	UF : 1, UT : 1,		CONFIG : 'N U T, 0, 0, 0',
	X =   648.092  mm,	Y = -1312.832  mm,	Z =  1599.443  mm,
	W =   -41.810 deg,	P =   -20.894 deg,	R =   -21.724 deg
   GP2:
	UF : 0, UT : 1,
	J1=   180.000 deg,	J2=   -90.000 deg
};
P[708]{
   GP1:
	UF : 1, UT : 1,		CONFIG : 'N U T, 0, 0, 0',
	X =   973.093  mm,	Y =   -11.831  mm,	Z =  2176.445  mm,
	W =     -.010 deg,	P =   -45.000 deg,	R =     0.000 deg
   GP2:
	UF : 0, UT : 1,
	J1=   180.000 deg,	J2=    90.000 deg
};
P[709]{
   GP1:
	UF : 1, UT : 1,		CONFIG : 'N U T, 0, 0, 0',
	X =  1331.092  mm,	Y =   987.169  mm,	Z =  1342.444  mm,
	W =     -.010 deg,	P =    45.000 deg,	R =   -90.000 deg
   GP2:
	UF : 0, UT : 1,
	J1=   180.000 deg,	J2=    90.000 deg
};
P[710]{
   GP1:
	UF : 1, UT : 1,		CONFIG : 'N U T, 0, 0, 0',
	X =  1864.092  mm,	Y =  1212.638  mm,	Z =  1342.445  mm,
	W =    44.958 deg,	P =    -2.212 deg,	R =     2.229 deg
   GP2:
	UF : 0, UT : 1,
	J1=   180.000 deg,	J2=    90.000 deg
};
P[711]{
   GP1:
	UF : 1, UT : 1,		CONFIG : 'N U T, 0, 0, 0',
	X =  1940.973  mm,	Y =  1347.132  mm,	Z =  1061.188  mm,
	W =    41.277 deg,	P =    19.800 deg,	R =   -21.086 deg
   GP2:
	UF : 0, UT : 1,
	J1=   180.000 deg,	J2=    90.000 deg
};
P[712]{
   GP1:
	UF : 1, UT : 1,		CONFIG : 'N U T, 0, 0, 0',
	X =  1901.875  mm,	Y =  1465.160  mm,	Z =  1036.238  mm,
	W =    41.263 deg,	P =    19.805 deg,	R =   -17.225 deg
   GP2:
	UF : 1, UT : 1,
	J1=   180.000 deg,	J2=    90.000 deg
};
P[713]{
   GP1:
	UF : 1, UT : 1,		CONFIG : 'N U T, 0, 0, 0',
	X =  1934.116  mm,	Y =  1464.614  mm,	Z =  1037.732  mm,
	W =    41.277 deg,	P =    19.801 deg,	R =   -17.230 deg
   GP2:
	UF : 1, UT : 1,
	J1=   180.000 deg,	J2=    90.000 deg
};
P[714]{
   GP1:
	UF : 1, UT : 1,		CONFIG : 'N U T, 0, 0, 0',
	X =  1965.909  mm,	Y =  1468.963  mm,	Z =  1032.171  mm,
	W =    41.272 deg,	P =    19.803 deg,	R =   -17.223 deg
   GP2:
	UF : 1, UT : 1,
	J1=   180.000 deg,	J2=    90.000 deg
};
P[715]{
   GP1:
	UF : 1, UT : 1,		CONFIG : 'N U T, 0, 0, 0',
	X =  1996.605  mm,	Y =  1480.121  mm,	Z =  1030.618  mm,
	W =    41.277 deg,	P =    19.801 deg,	R =     6.735 deg
   GP2:
	UF : 1, UT : 1,
	J1=   180.000 deg,	J2=    90.000 deg
};
P[716]{
   GP1:
	UF : 1, UT : 1,		CONFIG : 'N U T, 0, 0, 0',
	X =  1999.792  mm,	Y =  1488.994  mm,	Z =  1027.439  mm,
	W =    43.863 deg,	P =    11.272 deg,	R =    16.919 deg
   GP2:
	UF : 1, UT : 1,
	J1=   180.000 deg,	J2=    90.000 deg
};
P[717]{
   GP1:
	UF : 1, UT : 1,		CONFIG : 'N U T, 0, 0, 0',
	X =  2007.580  mm,	Y =  1422.903  mm,	Z =  1059.661  mm,
	W =    44.305 deg,	P =     8.850 deg,	R =     3.803 deg
   GP2:
	UF : 1, UT : 1,
	J1=   180.000 deg,	J2=    90.000 deg
};
P[718]{
   GP1:
	UF : 1, UT : 1,		CONFIG : 'N U T, 0, 0, 0',
	X =  1864.092  mm,	Y =  1212.638  mm,	Z =  1342.444  mm,
	W =    44.958 deg,	P =    -2.212 deg,	R =     2.229 deg
   GP2:
	UF : 0, UT : 1,
	J1=   180.000 deg,	J2=    90.000 deg
};
P[729]{
   GP1:
	UF : 1, UT : 1,		CONFIG : 'F U T, 0, 0, 0',
	X =   818.947  mm,	Y =   972.802  mm,	Z =  1108.910  mm,
	W =    50.730 deg,	P =      .639 deg,	R =   -51.736 deg
   GP2:
	UF : 1, UT : 1,
	J1=   180.000 deg,	J2=   150.000 deg
};
P[730]{
   GP1:
	UF : 1, UT : 1,		CONFIG : 'F U T, 0, 0, 0',
	X =  1078.589  mm,	Y =   991.016  mm,	Z =  1063.910  mm,
	W =    50.730 deg,	P =      .639 deg,	R =   -51.736 deg
   GP2:
	UF : 1, UT : 1,
	J1=   180.000 deg,	J2=   150.000 deg
};
P[731]{
   GP1:
	UF : 1, UT : 1,		CONFIG : 'F U T, 0, 0, 0',
	X =  1104.853  mm,	Y =  1006.203  mm,	Z =  1025.639  mm,
	W =    44.130 deg,	P =    -6.203 deg,	R =   -51.549 deg
   GP2:
	UF : 1, UT : 1,
	J1=   180.000 deg,	J2=   150.000 deg
};
P[732]{
   GP1:
	UF : 1, UT : 1,		CONFIG : 'F U T, 0, 0, 0',
	X =  1114.844  mm,	Y =  1000.704  mm,	Z =  1027.080  mm,
	W =    43.014 deg,	P =    -7.268 deg,	R =   -34.946 deg
   GP2:
	UF : 1, UT : 1,
	J1=   180.000 deg,	J2=   150.000 deg
};
P[733]{
   GP1:
	UF : 1, UT : 1,		CONFIG : 'F U T, 0, 0, 0',
	X =  1125.597  mm,	Y =   997.219  mm,	Z =  1027.206  mm,
	W =    42.651 deg,	P =   -14.126 deg,	R =   -20.722 deg
   GP2:
	UF : 1, UT : 1,
	J1=   180.000 deg,	J2=   150.000 deg
};
P[734]{
   GP1:
	UF : 1, UT : 1,		CONFIG : 'F U T, 0, 0, 0',
	X =  1138.321  mm,	Y =   996.177  mm,	Z =  1027.210  mm,
	W =    42.651 deg,	P =   -14.126 deg,	R =   -27.080 deg
   GP2:
	UF : 1, UT : 1,
	J1=   180.000 deg,	J2=   150.000 deg
};
P[735]{
   GP1:
	UF : 1, UT : 1,		CONFIG : 'F U T, 0, 0, 0',
	X =  1090.032  mm,	Y =   963.970  mm,	Z =  1058.684  mm,
	W =    50.535 deg,	P =   -23.426 deg,	R =   -25.981 deg
   GP2:
	UF : 1, UT : 1,
	J1=   180.000 deg,	J2=   150.000 deg
};
P[736]{
   GP1:
	UF : 1, UT : 1,		CONFIG : 'F U T, 0, 0, 0',
	X =   866.460  mm,	Y =   968.970  mm,	Z =  1058.684  mm,
	W =    50.535 deg,	P =   -23.426 deg,	R =   -25.981 deg
   GP2:
	UF : 1, UT : 1,
	J1=   180.000 deg,	J2=   150.000 deg
};
P[737]{
   GP1:
	UF : 1, UT : 1,		CONFIG : 'F U T, 0, 0, 0',
	X =   866.460  mm,	Y =   968.969  mm,	Z =  1794.399  mm,
	W =    50.535 deg,	P =   -23.425 deg,	R =   -25.981 deg
   GP2:
	UF : 1, UT : 1,
	J1=   180.000 deg,	J2=   150.000 deg
};
P[749]{
   GP1:
	UF : 1, UT : 1,		CONFIG : 'N U B, 0, 0, 0',
	X =   361.637  mm,	Y =   -13.715  mm,	Z =  2427.062  mm,
	W =     -.019 deg,	P =   -39.997 deg,	R =      .013 deg
   GP2:
	UF : 1, UT : 1,
	J1=   100.000 deg,	J2=   -90.000 deg
};
P[750]{
   GP1:
	UF : 1, UT : 1,		CONFIG : 'N U T, 0, 0, 0',
	X =   345.640  mm,	Y = -1572.170  mm,	Z =  1050.335  mm,
	W =    56.087 deg,	P =     8.668 deg,	R =   -95.934 deg
   GP2:
	UF : 1, UT : 1,
	J1=   100.000 deg,	J2=   -90.000 deg
};
P[751]{
   GP1:
	UF : 1, UT : 1,		CONFIG : 'N U T, 0, 0, -1',
	X =  2515.039  mm,	Y = -1508.170  mm,	Z =  1050.334  mm,
	W =   -50.284 deg,	P =   -30.325 deg,	R =    67.097 deg
   GP2:
	UF : 0, UT : 1,
	J1=   100.000 deg,	J2=   -90.000 deg
};
P[752]{
   GP1:
	UF : 1, UT : 1,		CONFIG : 'N U T, 0, 0, 0',
	X =  2788.736  mm,	Y = -1483.274  mm,	Z =   933.541  mm,
	W =   -37.771 deg,	P =   -31.405 deg,	R =    42.828 deg
   GP2:
	UF : 1, UT : 1,
	J1=   100.000 deg,	J2=   -90.000 deg
};
P[753]{
   GP1:
	UF : 1, UT : 1,		CONFIG : 'N U T, 0, 0, 0',
	X =  2790.127  mm,	Y = -1512.097  mm,	Z =   933.343  mm,
	W =   -37.782 deg,	P =   -31.394 deg,	R =    42.842 deg
   GP2:
	UF : 1, UT : 1,
	J1=   100.000 deg,	J2=   -90.000 deg
};
P[754]{
   GP1:
	UF : 1, UT : 1,		CONFIG : 'N U T, 0, 0, 0',
	X =  2777.828  mm,	Y = -1541.019  mm,	Z =   932.405  mm,
	W =   -42.870 deg,	P =   -22.985 deg,	R =    39.985 deg
   GP2:
	UF : 1, UT : 1,
	J1=   100.000 deg,	J2=   -90.000 deg
};
P[755]{
   GP1:
	UF : 1, UT : 1,		CONFIG : 'N U T, 0, 0, 0',
	X =  2762.396  mm,	Y = -1555.396  mm,	Z =   929.477  mm,
	W =   -45.718 deg,	P =   -14.892 deg,	R =    35.274 deg
   GP2:
	UF : 1, UT : 1,
	J1=   100.000 deg,	J2=   -90.000 deg
};
P[756]{
   GP1:
	UF : 1, UT : 1,		CONFIG : 'N U T, 0, 0, 0',
	X =  2731.844  mm,	Y = -1574.335  mm,	Z =   920.084  mm,
	W =   -45.718 deg,	P =   -14.891 deg,	R =    30.406 deg
   GP2:
	UF : 1, UT : 1,
	J1=   100.000 deg,	J2=   -90.000 deg
};
P[757]{
   GP1:
	UF : 1, UT : 1,		CONFIG : 'N U T, 0, 0, 0',
	X =  2725.103  mm,	Y = -1575.819  mm,	Z =   919.847  mm,
	W =   -45.718 deg,	P =   -14.891 deg,	R =    18.309 deg
   GP2:
	UF : 1, UT : 1,
	J1=   100.000 deg,	J2=   -90.000 deg
};
P[758]{
   GP1:
	UF : 1, UT : 1,		CONFIG : 'N U T, 0, 0, 0',
	X =  2712.522  mm,	Y = -1579.347  mm,	Z =   916.110  mm,
	W =   -45.718 deg,	P =   -14.891 deg,	R =     6.077 deg
   GP2:
	UF : 1, UT : 1,
	J1=   100.000 deg,	J2=   -90.000 deg
};
P[759]{
   GP1:
	UF : 1, UT : 1,		CONFIG : 'N U T, 0, 0, 0',
	X =  2684.760  mm,	Y = -1581.022  mm,	Z =   910.051  mm,
	W =   -45.718 deg,	P =   -14.891 deg,	R =     6.077 deg
   GP2:
	UF : 1, UT : 1,
	J1=   100.000 deg,	J2=   -90.000 deg
};
P[760]{
   GP1:
	UF : 1, UT : 1,		CONFIG : 'N U T, 0, 0, 0',
	X =  2624.684  mm,	Y = -1545.568  mm,	Z =  1157.185  mm,
	W =   -45.531 deg,	P =     6.252 deg,	R =    32.963 deg
   GP2:
	UF : 0, UT : 1,
	J1=   100.000 deg,	J2=   -90.000 deg
};
P[761]{
   GP1:
	UF : 1, UT : 1,		CONFIG : 'N U T, 0, 0, 0',
	X =   619.684  mm,	Y = -1545.568  mm,	Z =  1157.185  mm,
	W =   -45.531 deg,	P =     6.252 deg,	R =    32.963 deg
   GP2:
	UF : 0, UT : 1,
	J1=   100.000 deg,	J2=   -90.000 deg
};
P[771]{
   GP1:
	UF : 1, UT : 1,		CONFIG : 'N U B, 0, 0, 0',
	X =   361.637  mm,	Y =   -13.715  mm,	Z =  2427.062  mm,
	W =     -.019 deg,	P =   -39.997 deg,	R =      .013 deg
   GP2:
	UF : 1, UT : 1,
	J1=    90.000 deg,	J2=    90.000 deg
};
P[772]{
   GP1:
	UF : 1, UT : 1,		CONFIG : 'N U T, 0, 0, 0',
	X =  1600.281  mm,	Y =  1476.125  mm,	Z =  1082.764  mm,
	W =    44.983 deg,	P =     1.340 deg,	R =    -4.979 deg
   GP2:
	UF : 0, UT : 1,
	J1=    90.000 deg,	J2=    90.000 deg
};
P[773]{
   GP1:
	UF : 1, UT : 1,		CONFIG : 'N U T, 0, 0, 0',
	X =  2541.394  mm,	Y =  1548.125  mm,	Z =  1070.592  mm,
	W =    21.780 deg,	P =   -40.404 deg,	R =   -29.962 deg
   GP2:
	UF : 0, UT : 1,
	J1=    95.000 deg,	J2=    90.000 deg
};
P[774]{
   GP1:
	UF : 1, UT : 1,		CONFIG : 'N U T, 0, 0, 0',
	X =  2674.298  mm,	Y =  1497.536  mm,	Z =  1070.592  mm,
	W =    15.908 deg,	P =   -31.536 deg,	R =   -26.500 deg
   GP2:
	UF : 0, UT : 1,
	J1=    95.000 deg,	J2=    90.000 deg
};
P[775]{
   GP1:
	UF : 1, UT : 1,		CONFIG : 'N U T, 0, 0, 0',
	X =  2833.414  mm,	Y =  1483.559  mm,	Z =   885.495  mm,
	W =     1.862 deg,	P =   -42.072 deg,	R =    -2.894 deg
   GP2:
	UF : 1, UT : 1,
	J1=    95.000 deg,	J2=    90.000 deg
};
P[776]{
   GP1:
	UF : 1, UT : 1,		CONFIG : 'N U T, 0, 0, 0',
	X =  2833.081  mm,	Y =  1508.177  mm,	Z =   884.362  mm,
	W =     1.851 deg,	P =   -42.070 deg,	R =    -2.890 deg
   GP2:
	UF : 1, UT : 1,
	J1=    95.000 deg,	J2=    90.000 deg
};
P[777]{
   GP1:
	UF : 1, UT : 1,		CONFIG : 'N U T, 0, 0, 0',
	X =  2826.705  mm,	Y =  1541.371  mm,	Z =   879.685  mm,
	W =    47.457 deg,	P =    -2.512 deg,	R =   -28.093 deg
   GP2:
	UF : 1, UT : 1,
	J1=    95.000 deg,	J2=    90.000 deg
};
P[778]{
   GP1:
	UF : 1, UT : 1,		CONFIG : 'N U T, 0, 0, 0',
	X =  2808.617  mm,	Y =  1556.143  mm,	Z =   878.386  mm,
	W =    47.469 deg,	P =    -2.511 deg,	R =   -28.096 deg
   GP2:
	UF : 1, UT : 1,
	J1=    95.000 deg,	J2=    90.000 deg
};
P[779]{
   GP1:
	UF : 1, UT : 1,		CONFIG : 'N U T, 0, 0, 0',
	X =  2772.622  mm,	Y =  1570.522  mm,	Z =   877.279  mm,
	W =    47.469 deg,	P =    -2.511 deg,	R =   -28.096 deg
   GP2:
	UF : 1, UT : 1,
	J1=    95.000 deg,	J2=    90.000 deg
};
P[780]{
   GP1:
	UF : 1, UT : 1,		CONFIG : 'N U T, 0, 0, 0',
	X =  2766.040  mm,	Y =  1572.698  mm,	Z =   875.804  mm,
	W =    46.964 deg,	P =     8.281 deg,	R =   -26.942 deg
   GP2:
	UF : 1, UT : 1,
	J1=    95.000 deg,	J2=    90.000 deg
};
P[781]{
   GP1:
	UF : 1, UT : 1,		CONFIG : 'N U T, 0, 0, 0',
	X =  2756.734  mm,	Y =  1575.818  mm,	Z =   872.094  mm,
	W =    47.296 deg,	P =    13.421 deg,	R =   -20.078 deg
   GP2:
	UF : 1, UT : 1,
	J1=    94.995 deg,	J2=    90.000 deg
};
P[782]{
   GP1:
	UF : 1, UT : 1,		CONFIG : 'N U T, 0, 0, 0',
	X =  2725.010  mm,	Y =  1574.875  mm,	Z =   871.699  mm,
	W =    46.312 deg,	P =    12.118 deg,	R =   -20.583 deg
   GP2:
	UF : 1, UT : 1,
	J1=    95.000 deg,	J2=    90.000 deg
};
P[783]{
   GP1:
	UF : 1, UT : 1,		CONFIG : 'N U T, 0, 0, 0',
	X =  2601.214  mm,	Y =  1517.756  mm,	Z =  1073.770  mm,
	W =    42.689 deg,	P =    16.599 deg,	R =   -42.374 deg
   GP2:
	UF : 0, UT : 1,
	J1=    95.000 deg,	J2=    90.000 deg
};
P[784]{
   GP1:
	UF : 1, UT : 1,		CONFIG : 'N U T, 0, 0, 0',
	X =  1497.214  mm,	Y =  1517.756  mm,	Z =  1073.770  mm,
	W =    42.689 deg,	P =    16.599 deg,	R =   -42.374 deg
   GP2:
	UF : 0, UT : 1,
	J1=    95.000 deg,	J2=    90.000 deg
};
/END
